# B&R Automation Studio project PvJson_Sample
Automation Studio 6.1.0.62; technology packages: OpcUaCs 6.0.0

## Configuration ArSim

CPU PC_any, AutomationRuntime 6.2.1, Build 11.3.0, Vc 6.0.0

### Task classes (Cpu.sw)
```
Cyclic#4:
  PvJsonDemo <- PvJsonDemo.prg
  DemoTask <- DemoTask.prg
Binaries: udbdef, sysconf, iomap, ashwd, asfw, arconfig, ashwac
Libraries: FileIO, sys_lib, astime, runtime, ArCert, AsBrStr, PvJson
```

### Hardware
```
PC : PC_any v1.1.2.0 (OrderNumber=PC)
  ConfigurationID = PvJson_Sample_ArSim
  FileDevice1
  FileDeviceName1 = PvJson
  FileDevicePath1 = USER_PATH
  ActivateWebServer = 1
  ActivateSdm = 1
```

### BRRole.brrole - PC/AccessAndSecurity/UserRoleSystem/BRRole.brrole
```
Element BR_Anonymous (Type=BRRole)
Element BR_Engineer (Type=BRRole)
Element BR_Observer (Type=BRRole)
Element BR_SafetyAdmin (Type=BRRole)
Element BR_SecurityAdmin (Type=BRRole)
```

## Logical view

Binary libraries used (declarations not repeated): operator, runtime, astime, AsIecCon, ArCert, FileIO, sys_lib, AsBrStr, PvJson 4.73.0


### Program Logical/PvJsonDemo (IEC)

#### Variables.var
```iecst
VAR
	JsonSerializer_0 : JsonSerializer;
	JsonParser_0 : JsonParser;
END_VAR
```

#### Main.st
```iecst
PROGRAM _INIT
	(* Insert code here *)
	JsonSerializer_0.Enable := TRUE;
	JsonParser_0.Enable 	:= TRUE;
END_PROGRAM

PROGRAM _CYCLIC

	// JsonSerializer_0.Execute ---> Set it using watch to test the functionality
	JsonSerializer_0.PVname := ADR('DemoTask:DemoVar');
	JsonSerializer_0.FileDevice := ADR('PvJson'); //Defined at CPU config. It's pointing to C:\Temp\PvJson
	JsonSerializer_0.FileName := ADR('DemoVar.json');
	JsonSerializer_0();

	//JsonParser_0.Execute ---> Set it using watch to test the functionality
	JsonParser_0.FileDevice := ADR('PvJson');
	JsonParser_0.FileName 	:= ADR('DemoVar.json');
	JsonParser_0();
END_PROGRAM

PROGRAM _EXIT
	(* Insert code here *)
	JsonSerializer_0(Enable := FALSE);
	JsonParser_0(Enable := FALSE);
END_PROGRAM
```

### Program Logical/DemoTask (IEC)

#### Types.typ
```iecst
TYPE
	DemoStruct_type : 	STRUCT
		MyUsint : USINT;
		MyRealArray : ARRAY[-5..5]OF REAL;
		MyString : STRING[80];
		MyUnicodeString : WSTRING[80];
	END_STRUCT;
END_TYPE
```

#### Variables.var
```iecst
VAR
	DemoVar : DemoStruct_type;
	UnicodeMessage : ARRAY[0..80] OF UINT;
END_VAR
```

#### Main.st
```iecst
PROGRAM _INIT
	//https://apps.timwhitlock.info/unicode/inspect?s=%D0%9F%D1%80%D0%B8%D0%B2%D0%B5%D1%82
	UnicodeMessage[0] := 1055;
	UnicodeMessage[1] := 1088;
	UnicodeMessage[2] := 1080;
	UnicodeMessage[3] := 1074;
	UnicodeMessage[4] := 1077;
	UnicodeMessage[5] := 1090;
	brsmemcpy(ADR(DemoVar.MyUnicodeString),ADR(UnicodeMessage),MIN(SIZEOF(DemoVar.MyUnicodeString),SIZEOF(UnicodeMessage)));

	DemoVar.MyString := 'This is a demo string';
	DemoVar.MyUsint := 58;
	DemoVar.MyRealArray[-5] := -5.5;
	DemoVar.MyRealArray[-4] := -4.4;
	DemoVar.MyRealArray[-3] := -3.3;
	DemoVar.MyRealArray[-2] := -2.2;
	DemoVar.MyRealArray[-1] := -1.1;
	DemoVar.MyRealArray[0] 	:= 0;
	DemoVar.MyRealArray[1] 	:= 1.1;
	DemoVar.MyRealArray[2] 	:= 2.2;
	DemoVar.MyRealArray[3] 	:= 3.3;
	DemoVar.MyRealArray[4] 	:= 4.4;
	DemoVar.MyRealArray[5] 	:= 5.5;
END_PROGRAM

PROGRAM _CYCLIC
	(* Insert code here *)

END_PROGRAM

PROGRAM _EXIT
	(* Insert code here *)

END_PROGRAM
```

Listed in the project but not available here: Logical/Global.typ, Logical/Global.var
